FUNCTION VeranderLicht : VerkeerslichtStatus
VAR_INPUT
	StoplichtWissel	: VerkeerslichtStatus;
END_VAR


CASE StoplichtWissel OF
    VerkeerslichtStatus.Rood:
        VeranderLicht := VerkeerslichtStatus.Groen;   // Van Rood naar Groen
		
    VerkeerslichtStatus.Groen:
        VeranderLicht := VerkeerslichtStatus.Geel;  // Van Groen naar Geel
		
    VerkeerslichtStatus.Geel:
        VeranderLicht := VerkeerslichtStatus.Rood;    // Van Geel naar Rood
		
ELSE
    VeranderLicht := VerkeerslichtStatus.Rood;      // bij default moet het naar Rood
END_CASE

END_FUNCTION

(* stored: Version 1.1.0.1, ProductVersion 3.1.4024.12
   POU VeranderLicht: Id {415282d1-ffdf-458e-b9ba-dbf4956d2277}, SpecialFunc None *)
